(* PLC project EEDOMUS_TPL, Actility iec61131 1.0.28, author Laurent Nicq *)
(* stored: creationDateTime 2013-07-16T14:50:58, version 1.0.1, modificationDateTime 2013-09-10T17:36:39 *)

PROGRAM rules_template
  VAR
    EE_Rule_0000_Name : STRING := 'Rule_0000';
    EE_Rule_0000_TS_Active : DT;  (* Time Stamp Last Activation *)
    EE_Rule_0000_TS_LastExec : DT;  (* Time Stamp Last Execution *)
    EE_Rule_0000_State : DINT;  (* 0: waiting for condition 1: executing *)
  END_VAR
  VAR_EXTERNAL
    EE_Rule_0000_Count_Exec : DINT;  (* Number of execution *)
    EE_Rule_0000_Active : BOOL;
    EE_Rule_0000_GLO_Var_00 : DINT;
    EE_Rule_0000_GLO_Var_01 : DINT;
    EE_Rule_0000_GLO_Var_02 : DINT;
  END_VAR
  VAR
    EE_Rule_0000_LOC_Var_00 : DINT := 0;  (* initial value for Debug only *)
    EE_Rule_0000_LOC_Var_01 : DINT := 1;  (* initial value for Debug only *)
    EE_Rule_0000_LOC_Var_02 : DINT := 2;  (* initial value for Debug only *)
    EE_Rule_0000_CAL_SINGLE_00 : STRING := 'SINGLE_00';  (* initial value for Debug only *)
    EE_Rule_0000_CAL_DAILY_00 : STRING := 'DAILY_00';  (* initial value for Debug only *)
    EE_Rule_0000_CAL_WEEKLY_00 : STRING := 'WEEKLY_00';  (* initial value for Debug only *)
    EE_Rule_0000_CAL_WEEKLY_Days_00 : DINT := 2#0111_1111;  (* initial value for Debug only. Bit0: Sunday Bit1: Monday *)
    EE_Rule_0000_CAL_Daily_Start_00 : TOD := TOD#11:55:00;  (* Start Time for Daily Calendar *)
    EE_Rule_0000_CAL_Daily_Stop_00 : TOD := TOD#19:15:00;  (* Stop Time for Daily Calendar *)
    EE_Rule_0000_CAL_Weekly_Start_00 : TOD := TOD#12:20:00;  (* StartTime for Weekly Calendar *)
    EE_Rule_0000_CAL_Weekly_Stop_00 : TOD := TOD#18:20:00;  (* Stop Time for Weekly Calendar *)
  END_VAR
  VAR_EXTERNAL
    EE_Rule_GLOBAL_Day_Phase_00 : TOD;  (* Day Phase calculated in an other POU *)
    EE_Rule_GLOBAL_Day_Phase_01 : TOD;  (* Day Phase calculated in an other POU *)
    EE_Rule_GLOBAL_Day_Type : DINT;  (* 0: working 1: non-working 2: vacation *)
  END_VAR
  VAR
    EE_Rule_0000_Retrigger_TON : TON;
    EE_Rule_0000_Get_triggerET : TIME;  (* For debug and Test only *)
  END_VAR
  VAR_EXTERNAL
    EE_Rule_0000_Trigger_Wait : TIME;
  END_VAR
  VAR
    EE_Rule_0000_Trigger_Activate : BOOL;
    EE_Rule_0000_Trigger_Ready : BOOL;
  END_VAR

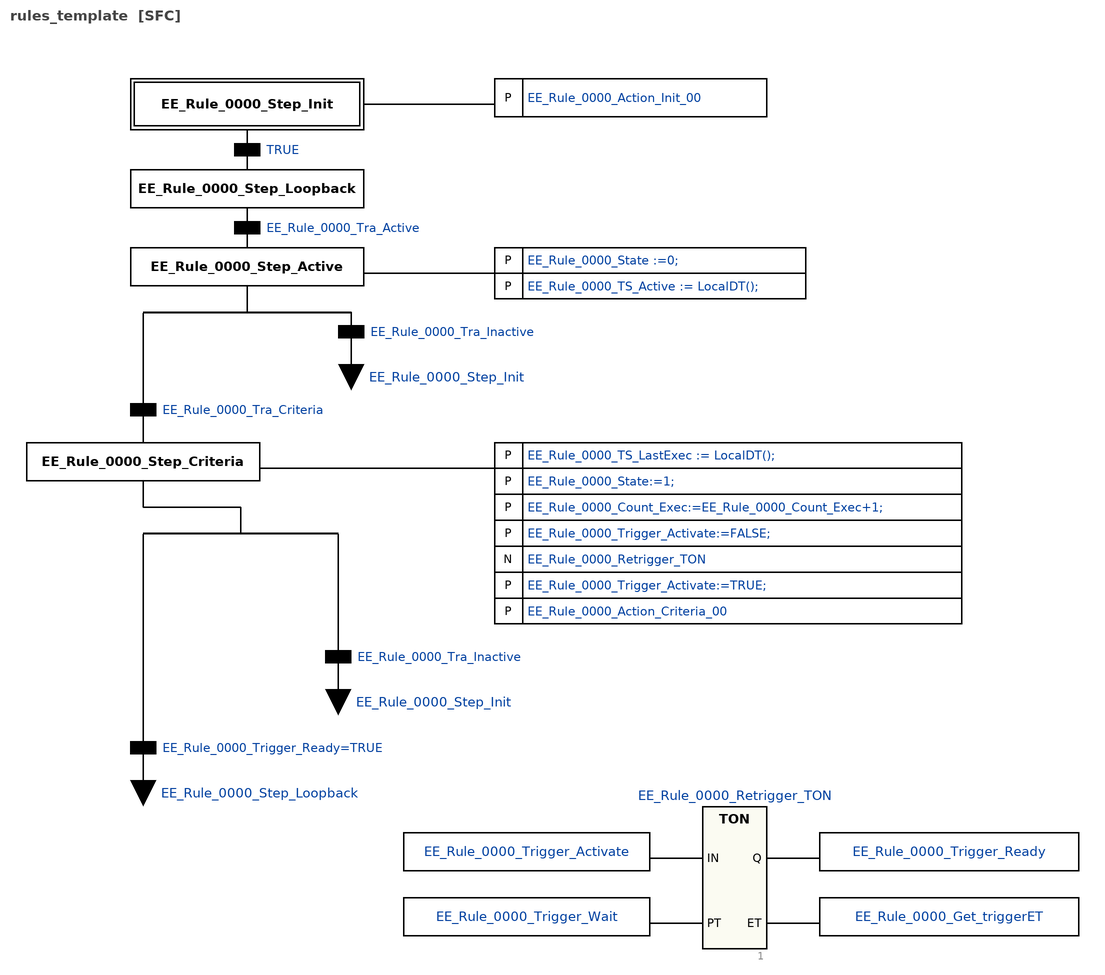
(* transition EE_Rule_0000_Tra_Timer *)
(* This transition is for all Timing and Calendar related conditions *)
(* If Timer are not used, leave it to TRUE *)
(* TRUE; *)
(* transition EE_Rule_0000_Tra_Criteria *)
(* This part of the transition is for Logical conditions in a Rule *)
(* If Criteria are not used, leave it to TRUE *)
(* TRUE; *)
(* This part transition is for all Timing and Calendar related conditions *)
(* If Timer are not used, leave it to TRUE *)
(* TRUE; *)
(* add an AND between the Time condition and Logical condition *)
INITIAL_STEP EE_Rule_0000_Step_Init:
  EE_Rule_0000_Action_Init_00(P);
  COMPUTE_FUNCTION_BLOCKS(S);
END_STEP
TRANSITION FROM (EE_Rule_0000_Step_Init, EE_Rule_0000_Step_Init, EE_Rule_0000_Step_Init) TO EE_Rule_0000_Step_Loopback
  := TRUE;
END_TRANSITION
STEP EE_Rule_0000_Step_Loopback:
END_STEP
TRANSITION FROM EE_Rule_0000_Step_Loopback TO EE_Rule_0000_Step_Active  (* EE_Rule_0000_Tra_Active *)
  := EE_Rule_0000_Active= TRUE;
END_TRANSITION
STEP EE_Rule_0000_Step_Active:
  EE_RULE_0000_STEP_ACTIVE_INLINE1(P);
  EE_RULE_0000_STEP_ACTIVE_INLINE2(P);
END_STEP
ACTION EE_RULE_0000_STEP_ACTIVE_INLINE1:
  EE_Rule_0000_State :=0;
END_ACTION
ACTION EE_RULE_0000_STEP_ACTIVE_INLINE2:
  EE_Rule_0000_TS_Active := LocalDT();
END_ACTION
TRANSITION FROM EE_Rule_0000_Step_Active TO EE_Rule_0000_Step_Criteria  (* EE_Rule_0000_Tra_Criteria *)
  := checkCalendarEvent( EE_Rule_0000_CAL_DAILY_00) OR checkCalendarEvent( EE_Rule_0000_CAL_WEEKLY_00);
END_TRANSITION
TRANSITION FROM EE_Rule_0000_Step_Active TO EE_Rule_0000_Step_Init  (* EE_Rule_0000_Tra_Inactive *)
  := EE_Rule_0000_Active= FALSE;
END_TRANSITION
STEP EE_Rule_0000_Step_Criteria:
  EE_RULE_0000_STEP_CRITERIA_INLINE3(P);
  EE_RULE_0000_STEP_CRITERIA_INLINE4(P);
  EE_RULE_0000_STEP_CRITERIA_INLINE5(P);
  EE_RULE_0000_STEP_CRITERIA_INLINE6(P);
  EE_Rule_0000_Retrigger_TON(N);
  EE_RULE_0000_STEP_CRITERIA_INLINE7(P);
  EE_Rule_0000_Action_Criteria_00(P);
END_STEP
ACTION EE_RULE_0000_STEP_CRITERIA_INLINE3:
  EE_Rule_0000_TS_LastExec := LocalDT();
END_ACTION
ACTION EE_RULE_0000_STEP_CRITERIA_INLINE4:
  EE_Rule_0000_State:=1;
END_ACTION
ACTION EE_RULE_0000_STEP_CRITERIA_INLINE5:
  EE_Rule_0000_Count_Exec:=EE_Rule_0000_Count_Exec+1;
END_ACTION
ACTION EE_RULE_0000_STEP_CRITERIA_INLINE6:
  EE_Rule_0000_Trigger_Activate:=FALSE;
END_ACTION
ACTION EE_RULE_0000_STEP_CRITERIA_INLINE7:
  EE_Rule_0000_Trigger_Activate:=TRUE;
END_ACTION
TRANSITION FROM EE_Rule_0000_Step_Criteria TO EE_Rule_0000_Step_Loopback
  := EE_Rule_0000_Trigger_Ready=TRUE;
END_TRANSITION
TRANSITION FROM EE_Rule_0000_Step_Criteria TO EE_Rule_0000_Step_Init  (* EE_Rule_0000_Tra_Inactive *)
  := EE_Rule_0000_Active= FALSE;
END_TRANSITION
ACTION COMPUTE_FUNCTION_BLOCKS:  (* blocks drawn on the SFC sheet *)
  EE_Rule_0000_Retrigger_TON(IN := EE_Rule_0000_Trigger_Activate, PT := EE_Rule_0000_Trigger_Wait);
  EE_Rule_0000_Trigger_Ready := EE_Rule_0000_Retrigger_TON.Q;
  EE_Rule_0000_Get_triggerET := EE_Rule_0000_Retrigger_TON.ET;
END_ACTION

ACTION EE_Rule_0000_Action_Init_00:
EE_Rule_0000_State:=-1;
(* Initialization of Variable and Function such as Calendar *)
newCalendarDailyEvent(  EE_Rule_0000_CAL_DAILY_00,
                        EE_Rule_0000_CAL_Daily_Start_00,
                        EE_Rule_0000_CAL_Daily_Stop_00,
                        1
                        );
newCalendarWeeklyEvent( EE_Rule_0000_CAL_WEEKLY_00,
                        EE_Rule_0000_CAL_Weekly_Start_00,
                        EE_Rule_0000_CAL_Weekly_Stop_00,
                        EE_Rule_0000_CAL_WEEKLY_Days_00
                        );
(* Multiple Actions can be created *)

              
END_ACTION

ACTION EE_Rule_0000_Action_Criteria_00:
(* Any USER action once the criteria and/or timer is matching goes here*)
(* there can be multiple separated Actions if necessary for code clarity *)
              
END_ACTION
END_PROGRAM

PROGRAM macros_template
  VAR_EXTERNAL
    EE_Macro_0000_Start : BOOL;
    EE_Macro_0000_Started : BOOL;
  END_VAR
  VAR
    EE_Macro_0000_Loop : BOOL;  (* indicates if Macro shall loopback *)
    EE_Macro_0000_Terminate : BOOL;  (* indicates if Macro shall terminate *)
    EE_Macro_0000_Name : STRING;  (* administrative, debug *)
    EE_Macro_0000_LOC_Wait_00 : TIME := T#5s;  (* Local wait time *)
    EE_Macro_0000_LOC_Wait_01 : TIME;
    EE_Macro_0000_LOC_Wait_02 : TIME;
  END_VAR
  VAR_EXTERNAL
    EE_Macro_0000_GLO_Wait_00 : TIME;  (* Global wait time *)
    EE_Macro_0000_GLO_Wait_01 : TIME;
  END_VAR
  VAR
    EE_Macro_0000_Random_Wait : TIME;
    EE_Macro_0000_WakeupTime : DT;
    EE_Macro_0000_WaitTime : TIME;
  END_VAR
  VAR_EXTERNAL
    EE_Macro_0000_GLO_OutBOOL_00 : BOOL;
    EE_Macro_0000_GLO_OutDINT_00 : DINT;
  END_VAR

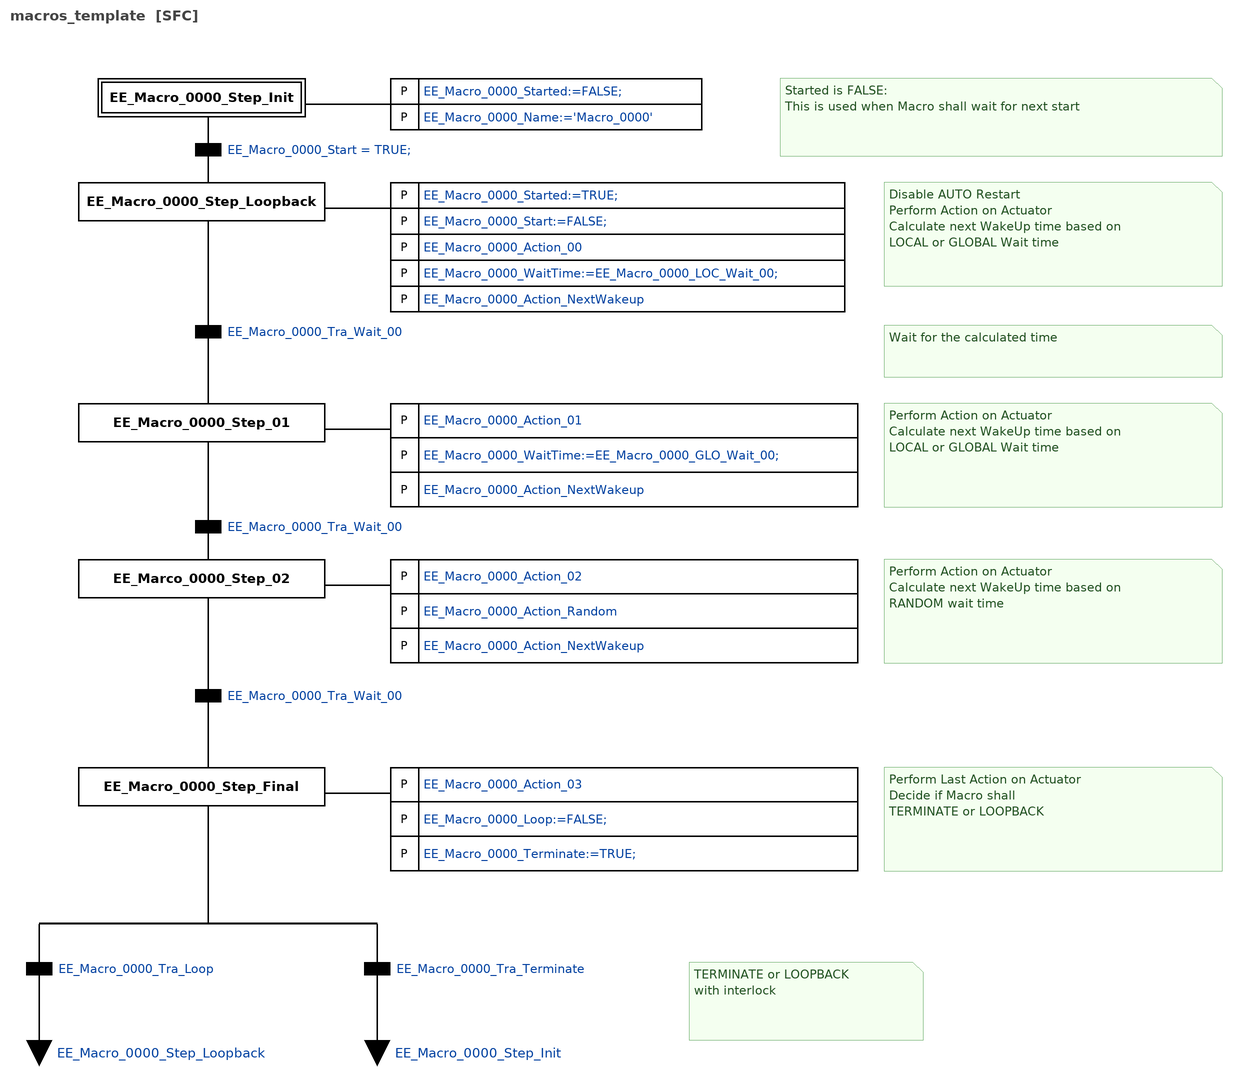
(* transition EE_Macro_0000_Tra_Wait_00 *)
(*If immediate action, set to TRUE*)
(*TRUE;*)
(* if time based *)
(* Started is FALSE:
This is used when Macro shall wait for next start *)
(* Disable AUTO Restart
Perform Action on Actuator
Calculate next WakeUp time based on
LOCAL or GLOBAL Wait time *)
(* Perform Action on Actuator
Calculate next WakeUp time based on
LOCAL or GLOBAL Wait time *)
(* Perform Last Action on Actuator
Decide if Macro shall
TERMINATE or LOOPBACK *)
(* Perform Action on Actuator
Calculate next WakeUp time based on
RANDOM wait time *)
(* TERMINATE or LOOPBACK
with interlock *)
(* Wait for the calculated time *)
INITIAL_STEP EE_Macro_0000_Step_Init:
  EE_MACRO_0000_STEP_INIT_INLINE1(P);
  EE_MACRO_0000_STEP_INIT_INLINE2(P);
END_STEP
ACTION EE_MACRO_0000_STEP_INIT_INLINE1:
  EE_Macro_0000_Started:=FALSE;
END_ACTION
ACTION EE_MACRO_0000_STEP_INIT_INLINE2:
  EE_Macro_0000_Name:='Macro_0000'
END_ACTION
TRANSITION FROM EE_Macro_0000_Step_Init TO EE_Macro_0000_Step_Loopback
  := EE_Macro_0000_Start = TRUE;
END_TRANSITION
STEP EE_Macro_0000_Step_Loopback:
  EE_MACRO_0000_STEP_LOOPBACK_INLINE3(P);
  EE_MACRO_0000_STEP_LOOPBACK_INLINE4(P);
  EE_Macro_0000_Action_00(P);
  EE_MACRO_0000_STEP_LOOPBACK_INLINE5(P);
  EE_Macro_0000_Action_NextWakeup(P);
END_STEP
ACTION EE_MACRO_0000_STEP_LOOPBACK_INLINE3:
  EE_Macro_0000_Started:=TRUE;
END_ACTION
ACTION EE_MACRO_0000_STEP_LOOPBACK_INLINE4:
  EE_Macro_0000_Start:=FALSE;
END_ACTION
ACTION EE_MACRO_0000_STEP_LOOPBACK_INLINE5:
  EE_Macro_0000_WaitTime:=EE_Macro_0000_LOC_Wait_00;
END_ACTION
TRANSITION FROM EE_Macro_0000_Step_Loopback TO EE_Macro_0000_Step_01  (* EE_Macro_0000_Tra_Wait_00 *)
  := LocalDT() >=EE_Macro_0000_WakeupTime;
END_TRANSITION
STEP EE_Macro_0000_Step_01:
  EE_Macro_0000_Action_01(P);
  EE_MACRO_0000_STEP_01_INLINE6(P);
  EE_Macro_0000_Action_NextWakeup(P);
END_STEP
ACTION EE_MACRO_0000_STEP_01_INLINE6:
  EE_Macro_0000_WaitTime:=EE_Macro_0000_GLO_Wait_00;
END_ACTION
TRANSITION FROM EE_Macro_0000_Step_01 TO EE_Marco_0000_Step_02  (* EE_Macro_0000_Tra_Wait_00 *)
  := LocalDT() >=EE_Macro_0000_WakeupTime;
END_TRANSITION
STEP EE_Marco_0000_Step_02:
  EE_Macro_0000_Action_02(P);
  EE_Macro_0000_Action_Random(P);
  EE_Macro_0000_Action_NextWakeup(P);
END_STEP
TRANSITION FROM EE_Marco_0000_Step_02 TO EE_Macro_0000_Step_Final  (* EE_Macro_0000_Tra_Wait_00 *)
  := LocalDT() >=EE_Macro_0000_WakeupTime;
END_TRANSITION
STEP EE_Macro_0000_Step_Final:
  EE_Macro_0000_Action_03(P);
  EE_MACRO_0000_STEP_FINAL_INLINE7(P);
  EE_MACRO_0000_STEP_FINAL_INLINE8(P);
END_STEP
ACTION EE_MACRO_0000_STEP_FINAL_INLINE7:
  EE_Macro_0000_Loop:=FALSE;
END_ACTION
ACTION EE_MACRO_0000_STEP_FINAL_INLINE8:
  EE_Macro_0000_Terminate:=TRUE;
END_ACTION
TRANSITION FROM EE_Macro_0000_Step_Final TO EE_Macro_0000_Step_Loopback  (* EE_Macro_0000_Tra_Loop *)
  := (EE_Macro_0000_Loop= TRUE) AND (EE_Macro_0000_Terminate= FALSE);
END_TRANSITION
TRANSITION FROM EE_Macro_0000_Step_Final TO EE_Macro_0000_Step_Init  (* EE_Macro_0000_Tra_Terminate *)
  := (EE_Macro_0000_Loop= FALSE) AND (EE_Macro_0000_Terminate= TRUE);
END_TRANSITION

ACTION EE_Macro_0000_Action_NextWakeup:
EE_Macro_0000_WakeupTime:= ADD_DT_TIME( LocalDT(), EE_Macro_0000_WaitTime);
              
END_ACTION

ACTION EE_Macro_0000_Action_Random:
(* Calculate a randon Wait Time *)
(* Example for Random between 2 and 10 sec *)
EE_Macro_0000_Random_Wait := DINT_TO_TIME( 2 + RAND (8) );
              
END_ACTION

ACTION EE_Macro_0000_Action_00:
(* Action to be performed on Actuators *)
EE_Macro_0000_GLO_OutBOOL_00:=TRUE;
EE_Macro_0000_GLO_OutDINT_00:=EE_Macro_0000_GLO_OutDINT_00+1;

              
END_ACTION

ACTION EE_Macro_0000_Action_01:
EE_Macro_0000_GLO_OutBOOL_00:=FALSE;
EE_Macro_0000_GLO_OutDINT_00:=EE_Macro_0000_GLO_OutDINT_00+1;
              
END_ACTION

ACTION EE_Macro_0000_Action_02:
EE_Macro_0000_GLO_OutBOOL_00:=TRUE;
EE_Macro_0000_GLO_OutDINT_00:=EE_Macro_0000_GLO_OutDINT_00+1;
              
END_ACTION

ACTION EE_Macro_0000_Action_03:
EE_Macro_0000_GLO_OutBOOL_00:=FALSE;
EE_Macro_0000_GLO_OutDINT_00:=EE_Macro_0000_GLO_OutDINT_00+1;
              
END_ACTION
END_PROGRAM

CONFIGURATION config
  RESOURCE Common_Resource ON PLC
    VAR_GLOBAL
      EE_Rule_0000_Active AT %IX0000 : BOOL := TRUE;  (* TRUE for Debug only *)
      EE_Rule_GLOBAL_Day_Phase_00 : TOD;
      EE_Rule_GLOBAL_Day_Phase_01 : TOD;
      EE_Rule_GLOBAL_Day_Type : DINT;
      EE_Rule_0000_Trigger_Wait : TIME := t#5s;
      EE_Rule_0000_GLO_Var_00 AT %IX0001 : DINT := 10;  (* Initial Value for Debug only *)
      EE_Rule_0000_GLO_Var_01 : DINT := 11;  (* Initial Value for Debug only *)
      EE_Rule_0000_GLO_Var_02 : DINT := 12;  (* Initial Value for Debug only *)
    END_VAR
    VAR_GLOBAL RETAIN
      EE_Rule_0000_Count_Exec AT %QX0000 : DINT;
    END_VAR
    VAR_GLOBAL
      EE_Macro_0000_Start : BOOL := TRUE;  (* Initial Value for Debug only *)
      EE_Macro_0000_Started : BOOL;
      EE_Macro_0000_GLO_Wait_00 : TIME := t#10s;
      EE_Macro_0000_GLO_Wait_01 : TIME;
      EE_Macro_0000_GLO_OutBOOL_00 : BOOL;
      EE_Macro_0000_GLO_OutDINT_00 : DINT;
    END_VAR
    TASK Trigger_Fast1(INTERVAL := t#100ms, PRIORITY := 0);
    TASK Trigger_Fast2(INTERVAL := t#200ms, PRIORITY := 0);
    TASK Trigger_Slow1(INTERVAL := t#1s, PRIORITY := 0);
    TASK Trigger_Slow2(INTERVAL := t#2s, PRIORITY := 0);
    TASK (PRIORITY := 0);
    PROGRAM Macro_0000 WITH Trigger_Slow1 : macros_template;
    PROGRAM Rule_0000 WITH Trigger_Slow1 : rules_template;
  END_RESOURCE
END_CONFIGURATION
